FUNCTION_BLOCK WatchDog
VAR_INPUT
END_VAR
VAR_OUTPUT
END_VAR
VAR
	Timer : TON;
	Enabled : BOOL;
	TimeSpan : TIME := T#1S;
END_VAR

Timer(IN:=Enabled, PT:=TimeSpan);

METHOD PUBLIC Disable : BOOL
VAR_INPUT
END_VAR
Enabled := FALSE;
THIS^();
END_METHOD

METHOD PUBLIC Enable
VAR_INPUT
	Duration : TIME;
END_VAR
TimeSpan := Duration;
Enabled := TRUE;
THIS^();
END_METHOD

PROPERTY PUBLIC isTriggered : BOOL
GET
THIS^();
isTriggered := Timer.Q;
END_GET
END_PROPERTY

METHOD PUBLIC Reset : BOOL
VAR_INPUT
END_VAR
Disable();
Enable(TimeSpan);
END_METHOD

END_FUNCTION_BLOCK

(* stored: Version 1.1.0.1, ProductVersion 3.1.4024.9
   POU WatchDog: Id {ed8665c8-6b19-4490-9b90-bc87be843128}, SpecialFunc None
   Method Disable: Id {95c6f188-0992-43c9-82e2-6d36d22c4078}
   Method Enable: Id {1c98ed3a-c063-40b2-aae9-6d0e5e1e579f}
   Property isTriggered: Id {3168c9cc-acc0-45d3-8b30-c08b41368388}
   Get Get: Id {f93bc7ce-82d4-4c5b-ae87-4cb91023bd70}
   Method Reset: Id {1847def5-837a-4668-a950-37ab8f07054e} *)
